FUNCTION_BLOCK EL3144
VAR
	_io : EL3xx4_Data;
	{attribute addProperty Name "WcState"}
	_wcState : WcStateInputToggle;
	{attribute addProperty Name "Info data"}
	_infoData : InfoDataAds;
END_VAR

PROPERTY IO : REFERENCE TO EL3xx4_Data
GET
IO REF= _io;
END_GET
END_PROPERTY

PROPERTY WcState : REFERENCE TO WcStateInputToggle
GET
WcState REF= _wcState;
END_GET
END_PROPERTY

END_FUNCTION_BLOCK

(* stored: Version 1.1.0.1, ProductVersion 3.1.4024.9
   POU EL3144: Id {d44d5fe3-75ef-0ff3-34db-fed1895b4e96}, SpecialFunc None
   Property IO: Id {b7072724-8073-0c65-3ea9-d138af83b58e}
   Get Get: Id {7095fa25-87f4-09e0-2abd-a99116d47d67}
   Property WcState: Id {d0b792a1-d7fe-015e-1fa9-f531d9b21d8c}
   Get Get: Id {904ec475-f824-08be-2dc7-b8773c60a3d2} *)
